// TIA Portal project "SORTING 1" (V15)
// Vorlageprojekt für das Buch mit Zielsystem S7-1200

(* hardware
DEVICE "S7-1200-Station_1"  S7-1200 Station
   slot 0: "Baugruppenträger_0"  Rack  V1.0
   slot 1: "PLC_1"  CPU 1211C DC/DC/DC  6ES7 211-1AE40-0XB0  V4.1
*)

// ===== PLC "PLC_1"  CPU 1211C DC/DC/DC =====

VAR_GLOBAL   // PLC tag table "Standard-Variablentabelle"
   "Tag_1" AT %A0.0 : Bool;
   "Tag_2" AT %E0.0 : Bool;
   "Tag_3" AT %E0.1 : Bool;
   "Tag_4" AT %Q0.2 : Bool;
   "Tag_5" AT %I0.2 : Bool;
   "Tag_6" AT %Q0.3 : Bool;
   "Tag_7" AT %Q0.4 : Bool;
   "Tag_8" AT %Q0.5 : Bool;
   "Tag_9" AT %I0.4 : Bool;
   "Tag_10" AT %Q0.1 : Bool;
   "Tag_11" AT %I0.6 : Bool;
   "Tag_12" AT %I0.3 : Bool;
   "Tag_13" AT %M0.0 : Bool;
   "Tag_14" AT %I1.0 : Bool;
   "Tag_15" AT %M1.0 : Bool;
   "Tag_16" AT %Q1.0 : Bool;
   "M1" AT %M0.1 : Bool;
   "SENSOR" AT %I10.2 : Bool;
   "BELT 6M" AT %Q10.0 : Bool;
   "START" AT %I10.0 : Bool;
   "PUSHER FRONT" AT %I10.4 : Bool;
   "M2" AT %M0.2 : Bool;
   "PUSHER" AT %Q10.2 : Bool;
   "BELT 2M" AT %Q10.1 : Bool;
   "STOP" AT %I10.1 : Bool;
END_VAR

FUNCTION "MHJ-PLC-Lab-Function-S71200" : Void   // FC9000, SCL
{ S7_Optimized_Access := 'TRUE' }
VERSION : 0.1
   VAR_TEMP
      rdTimeReturn : Int;
      outputTime : DTL;
      SyncVal : Byte;
      forVal : Int;
      forVal_2 : Int;
      Value : Byte;
   END_VAR
   VAR CONSTANT
      CompVal : Byte := 16#34;
      Value_01 : Byte := 16#11;
      Value_01_DW : DWord := 16#A165_D992;
      Value_02_DW : DWord := 16#58BE_4401;
   END_VAR
BEGIN

   #Value:=PEEK(area := 16#82,
        dbNumber := 0,
        byteOffset := 511);
   #Value := #Value + 1;

   POKE(area := 16#82,
        dbNumber := 0,
        byteOffset := 511,
        value := #Value);

   POKE(area:=16#81,
        dbNumber:=0,
        byteOffset:=1016,
        value:=#Value_01_DW);
   POKE(area := 16#81,
        dbNumber := 0,
        byteOffset := 1020,
        value := #Value_02_DW);

   POKE(area := 16#81,
        dbNumber := 0,
        byteOffset := 511,
        value := B#16#00);

   FOR #forVal := 0 TO 120 DO
       FOR #forVal_2:=0 TO 10 DO
           #rdTimeReturn:=RD_SYS_T(#outputTime);
           #rdTimeReturn := WR_SYS_T(#outputTime);
           #rdTimeReturn := RD_SYS_T(#outputTime);
           #rdTimeReturn := WR_SYS_T(#outputTime);
       END_FOR;
       #SyncVal:= PEEK(area := 16#81,
                      dbNumber := 0,
                      byteOffset := 511);
       IF #SyncVal = #CompVal THEN
          GOTO M_1;
       END_IF;
   END_FOR;
   RETURN;

   M_1:
   POKE(area := 16#81,
        dbNumber := 0,
        byteOffset := 511,
        value := B#16#0);
END_FUNCTION

ORGANIZATION_BLOCK "Main"   // OB1, LAD, ProgramCycle
TITLE = "Main Program Sweep (Cycle)"
{ S7_Optimized_Access := 'TRUE' }
VERSION : 0.1
   VAR_INPUT
      Initial_Call : Bool;   // Initial call of this OB
      Remanence : Bool;   // =True, if remanent data are available
   END_VAR
   VAR_TEMP   // added for the SCL form of the ladder/FBD networks
      _w1 : Bool;
   END_VAR
BEGIN

REGION Network 1: Konnektierungsbaustein für PLC-Lab
   // Im Netzwerk 1 wird der Konnektierungsbaustein für PLC-Lab aufgerufen.
   // Dieser Aufruf darf nicht entfernt werden!
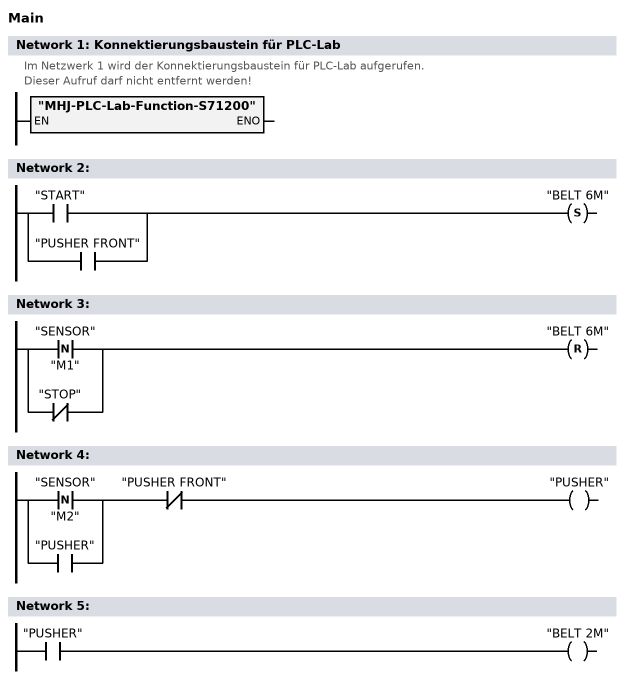
   RUNG wire#powerrail
      "MHJ-PLC-Lab-Function-S71200"()
   END_RUNG
   // the same network as SCL:
   "MHJ-PLC-Lab-Function-S71200"();
END_REGION

REGION Network 2
   RUNG wire#powerrail
      Contact( "START" )
      wire#w1
      S_Coil( "BELT 6M" )
   END_RUNG
   RUNG wire#powerrail
      Contact( "PUSHER FRONT" )
   END_RUNG wire#w1
   // the same network as SCL:
   IF "START" OR "PUSHER FRONT" THEN "BELT 6M" := TRUE; END_IF;
END_REGION

REGION Network 3
   RUNG wire#powerrail
      N_Contact(operand := "SENSOR", bit := "M1")
      wire#w1
      R_Coil( "BELT 6M" )
   END_RUNG
   RUNG wire#powerrail
      I_Contact( "STOP" )
   END_RUNG wire#w1
   // the same network as SCL:
   #_w1 := NOT "SENSOR" AND "M1";   // falling edge of "SENSOR"
   "M1" := "SENSOR";
   IF #_w1 OR NOT "STOP" THEN "BELT 6M" := FALSE; END_IF;
END_REGION

REGION Network 4
   RUNG wire#powerrail
      N_Contact(operand := "SENSOR", bit := "M2")
      wire#w1
      I_Contact( "PUSHER FRONT" )
      Coil( "PUSHER" )
   END_RUNG
   RUNG wire#powerrail
      Contact( "PUSHER" )
   END_RUNG wire#w1
   // the same network as SCL:
   #_w1 := NOT "SENSOR" AND "M2";   // falling edge of "SENSOR"
   "M2" := "SENSOR";
   "PUSHER" := (#_w1 OR "PUSHER") AND NOT "PUSHER FRONT";
END_REGION

REGION Network 5
   RUNG wire#powerrail
      Contact( "PUSHER" )
      Coil( "BELT 2M" )
   END_RUNG
   // the same network as SCL:
   "BELT 2M" := "PUSHER";
END_REGION
END_ORGANIZATION_BLOCK